Universal Robots PolyScope program: dev3_group1.urp

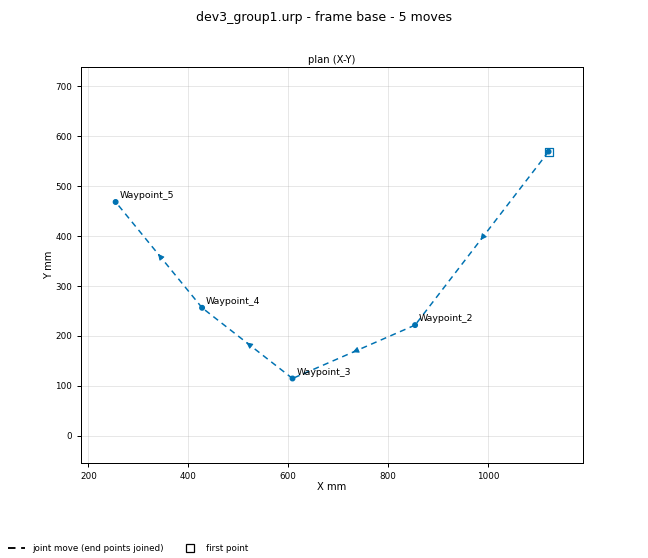
[picture p0: tool path of dev3_group1.urp in frame base, 5 of 5 moves have a stored position in this frame; points joined in program order, loops and branches not executed]
Program dev3_group1 (installation=default directory=/programs/usbdisk/Dev3_Group1 createdIn=5.11.10.1010502 lastSavedIn=5.11.10.1010502 robotSerialNumber=20225201339)
Calibrated DH parameters: a=[-0.000118, -0.339742, -0.555336, 0.000027, 0.000053, 0]; d=[0.180691, -465.540026, 499.223902, -33.510242, 0.119749, 0.115686]; alpha=[1.571428, -0.001093, 0.003977, 1.569316, -1.571413, 0]; deltaTheta=[0, 0.982125, 5.537749, -0.236695, 0, 0]
Robot Program (runOnlyOnce=false)
  MoveJ speed 60 deg/s, acceleration 80 deg/s^2 (useActiveTCP=true) feature=Base
    Waypoint Waypoint_1: TCP in base x=1121.493 y=569.203 z=781.726 mm, rx=-1.1036 ry=-1.1559 rz=0.9676 rad; joints [49.792, -128.485, -48.924, -8.583, 31.701, 16.419] deg; TCP offset x=-0.188 y=3.576 z=256.261 mm, rx=-0.0017 ry=3.1416 rz=0 rad
    Waypoint Waypoint_2: TCP in base x=854.123 y=221.714 z=781.694 mm, rx=-1.1036 ry=-1.156 rz=0.9677 rad; joints [47.643, -86.2, -104.489, 4.968, 33.826, 16.097] deg
    Waypoint Waypoint_3: TCP in base x=608.623 y=114.78 z=781.71 mm, rx=-1.1036 ry=-1.156 rz=0.9677 rad; joints [71.152, -53.068, -124.889, -19.475, 10.771, 28.425] deg
    Waypoint Waypoint_4: TCP in base x=427.526 y=256.379 z=781.687 mm, rx=-1.1035 ry=-1.1559 rz=0.9677 rad; joints [112.393, -62.422, -97.037, -193.991, 31.096, 185.485] deg
    Waypoint Waypoint_5: TCP in base x=254.365 y=468.316 z=781.671 mm, rx=-1.1036 ry=-1.1559 rz=0.9677 rad; joints [121.166, -84.393, -82.033, -188.34, 39.872, 187.03] deg
